{attribute 'GeneratedUsingTerminal: EL3141-0000-0016'}
{attribute addProperty BoxType "EL3141-0000-0016"}
{attribute addProperty Id "EtcSlaveTerminalBaseAI_StandardAT %I*AI_Standard_A8DF64E310WcStateAT %I*WcState_9091E0EB2InfoDataAT %I*InfoData_32EB74EA10"}
{attribute addProperty CRC "279820378"}
{attribute addProperty Size "22"}
TYPE EL3141_10ADB85A EXTENDS EtcSlaveTerminalBase :
STRUCT
	{attribute addProperty Name "AI_Standard"}
	AI_Standard : AI_Standard_A8DF64E3;
	{attribute addProperty Name "WcState"}
	WcState : WcState_9091E0EB;
	{attribute addProperty Name "InfoData"}
	InfoData : InfoData_32EB74EA;
END_STRUCT
END_TYPE

(* stored: Version 1.2.0.0, ProductVersion 3.1.4024.9
   DUT EL3141_10ADB85A: Id {23405e9a-6153-4475-982c-abb8e23a857f} *)
